(* IEC 61131-3 sources: Elmo_Master/test/Reports_Lasal/C78_20260807_publish_split_rebaseline (part 7) *)

END_FUNCTION

FUNCTION LMCControlCommandService::HandleAxisOwnershipPublishHomeReceipt
	VAR_INPUT
		AxisMask 	: UDINT;
		AdmissionToken 	: UDINT;
		OwnerGeneration 	: UDINT;
		ReportKind 	: UINT;
		ReportValue0 	: UDINT;
		ReportValue1 	: UDINT;
		ObservationCycle 	: UDINT;
	END_VAR
	VAR_OUTPUT
		Result 	: DINT;
	END_VAR

END_FUNCTION

FUNCTION LMCControlCommandService::PrepareAxisOwnershipPublishDecision
	VAR_INPUT
		AxisMask 	: UDINT;
		AdmissionToken 	: UDINT;
		OwnerGeneration 	: UDINT;
		ReportKind 	: UINT;
		ExpectedSession 	: UDINT;
		ExpectedSequence 	: UDINT;
		ExpectedCommandId 	: DINT;
		ExpectedReference 	: DINT;
		ExpectedAdmissionMode 	: DINT;
		ExpectedOwnerKind 	: DINT;
	END_VAR
	VAR_OUTPUT
		Result 	: DINT;
	END_VAR

END_FUNCTION
